TYPE ST_ITC_GroupCommands :
(**************************************************************************************
 * 	Application		:	BoxControl Framework
 *	Revision		:	$Revision: 404529 $
 *	Revision date	:	$Date: 2018-04-23 08:21:38 +0200 (Mo., 23 Apr 2018) $
 *	Last changed by	:	$Author: b7bolm $
 *	URL				:	$URL: http://almscdc.swisslog.com/repo/SWPD/Development/BoxControlFramework/20_Release/trunk/01_Software/BCF/BCF/JumpStart/20_Product/10_App/14_Groups/10_Lib/10_Conv/01_DUTs/ST_ITC_GroupCommands.TcDUT $
 *
 *	Purpose			:	Internal ITC group commands
 *
 * ------------------------------------------------------------------------------------
 *	Copyright Swisslog [IP AG], Switzerland. All rights reserved.
 * 
 * ------------------------------------------------------------------------------------
 *	
 * 	Revision History: 
 *
 * 	VERSION			DATE			INITIALS			DESCRIPTION
 *	0.1				01.01.2001		swl					Example
 *
 **************************************************************************************)
STRUCT
	Start					: BOOL; // Command: Start group 
	Stop					: BOOL; // Command: Stop group
	eMode					: E_PositionMode; // Command: Requested mode
	NoErrorReport			: BOOL; // Command: Send no error report
	StatusReport			: BOOL; // Command: Send StatusReport
	ControlReport			: BOOL; // command: Send ControlReport
END_STRUCT
END_TYPE

(* stored: Version 1.1.0.1, ProductVersion 3.1.4022.12
   DUT ST_ITC_GroupCommands: Id {ab13cbb4-fbd2-4dae-89ec-70eb83f2d7e5} *)
